// TIA Portal V16 export
// export: Created 2022-11-24T15:20:55.7439913Z, ExportSetting WithDefaults, DisplayName Totally Integrated Automation Portal, DisplayVersion V16 Update 6, DisplayName TIA Portal Version Control Interface, DisplayVersion V16 Update 2, DisplayName TIA Portal Openness, DisplayVersion V16 Update 6, DisplayName SINAMICS Startdrive Advanced, DisplayVersion V16 Update 5, DisplayName SINAMICS Startdrive G130, G150, S120, S150, SINAMICS MV, S210, DisplayVersion V16 Update 5, DisplayName SINAMICS Startdrive G110M, G120, G120C, G120D, G120P, G115D, DisplayVersion V16 Update 5, DisplayName STEP 7 Professional, DisplayVersion V16 Update 6, DisplayName STEP 7 Safety, DisplayVersion V16, DisplayName WinCC Advanced, DisplayVersion V16 Update 6
FUNCTION "FC62_PreStretchPGSAoutPWM" : Void   // FC62, LAD
{ S7_Optimized_Access := 'FALSE' }
AUTHOR : PaZan
VERSION : 0.1
// stored: AutoNumber false, IsIECCheckEnabled false, SetENOAutomatically false, UDAEnableTagReadback false
BEGIN

REGION Network 1: copy parameter for scale value % prestretch
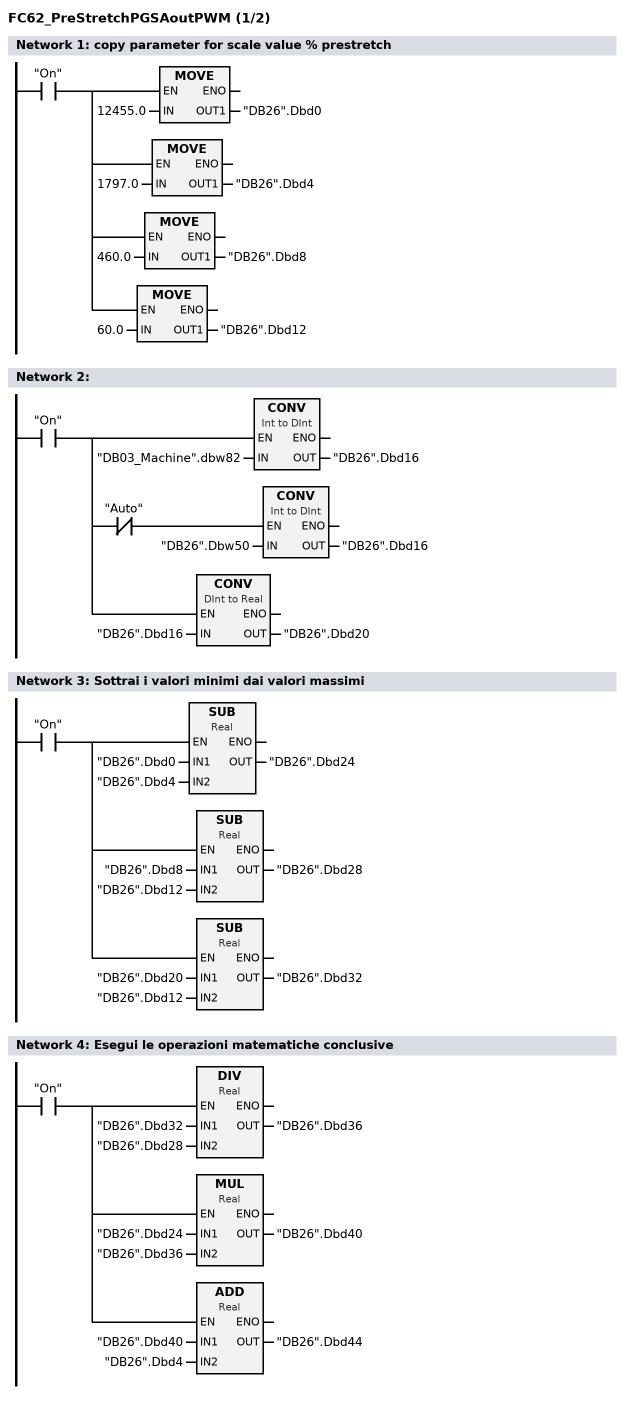
   RUNG wire#powerrail
      Contact( "On" )
      wire#w1
      { S7_GenerateENO := "TRUE" } Move(in := 12455.0, out1 => "DB26".Dbd0)
   END_RUNG
   RUNG wire#w1
      { S7_GenerateENO := "TRUE" } Move(in := 1797.0, out1 => "DB26".Dbd4)
   END_RUNG
   RUNG wire#w1
      { S7_GenerateENO := "TRUE" } Move(in := 460.0, out1 => "DB26".Dbd8)
   END_RUNG
   RUNG wire#w1
      { S7_GenerateENO := "TRUE" } Move(in := 60.0, out1 => "DB26".Dbd12)
   END_RUNG
   // the same network as SCL:
   IF "On" THEN
       "DB26".Dbd0 := 12455.0;
       "DB26".Dbd4 := 1797.0;
       "DB26".Dbd8 := 460.0;
       "DB26".Dbd12 := 60.0;
   END_IF;
END_REGION

REGION Network 2
   RUNG wire#powerrail
      Contact( "On" )
      wire#w1
      { S7_Templates := "[SrcType := Int, DestType := DInt]"; S7_GenerateENO := "TRUE" } Convert(in := "DB03_Machine".dbw82, out => "DB26".Dbd16)
   END_RUNG
   RUNG wire#w1
      I_Contact( "Auto" )
      { S7_Templates := "[SrcType := Int, DestType := DInt]"; S7_GenerateENO := "TRUE" } Convert(in := "DB26".Dbw50, out => "DB26".Dbd16)
   END_RUNG
   RUNG wire#w1
      { S7_Templates := "[SrcType := DInt, DestType := Real]"; S7_GenerateENO := "TRUE" } Convert(in := "DB26".Dbd16, out => "DB26".Dbd20)
   END_RUNG
   // the same network as SCL:
   IF "On" THEN "DB26".Dbd16 := INT_TO_DINT("DB03_Machine".dbw82); END_IF;
   IF "On" AND NOT "Auto" THEN "DB26".Dbd16 := INT_TO_DINT("DB26".Dbw50); END_IF;
   IF "On" THEN "DB26".Dbd20 := DINT_TO_REAL("DB26".Dbd16); END_IF;
END_REGION

REGION Network 3: Sottrai i valori minimi dai valori massimi
   RUNG wire#powerrail
      Contact( "On" )
      wire#w1
      { S7_Templates := "SrcType := Real"; S7_GenerateENO := "TRUE" } Sub(in1 := "DB26".Dbd0, in2 := "DB26".Dbd4, out => "DB26".Dbd24)
   END_RUNG
   RUNG wire#w1
      { S7_Templates := "SrcType := Real"; S7_GenerateENO := "TRUE" } Sub(in1 := "DB26".Dbd8, in2 := "DB26".Dbd12, out => "DB26".Dbd28)
   END_RUNG
   RUNG wire#w1
      { S7_Templates := "SrcType := Real"; S7_GenerateENO := "TRUE" } Sub(in1 := "DB26".Dbd20, in2 := "DB26".Dbd12, out => "DB26".Dbd32)
   END_RUNG
   // the same network as SCL:
   IF "On" THEN
       "DB26".Dbd24 := "DB26".Dbd0 - "DB26".Dbd4;
       "DB26".Dbd28 := "DB26".Dbd8 - "DB26".Dbd12;
       "DB26".Dbd32 := "DB26".Dbd20 - "DB26".Dbd12;
   END_IF;
END_REGION

REGION Network 4: Esegui le operazioni matematiche conclusive
   RUNG wire#powerrail
      Contact( "On" )
      wire#w1
      { S7_Templates := "SrcType := Real"; S7_GenerateENO := "TRUE" } Div(in1 := "DB26".Dbd32, in2 := "DB26".Dbd28, out => "DB26".Dbd36)
   END_RUNG
   RUNG wire#w1
      { S7_Templates := "SrcType := Real"; S7_GenerateENO := "TRUE" } Mul(in1 := "DB26".Dbd24, in2 := "DB26".Dbd36, out => "DB26".Dbd40)
   END_RUNG
   RUNG wire#w1
      { S7_Templates := "SrcType := Real"; S7_GenerateENO := "TRUE" } Add(in1 := "DB26".Dbd40, in2 := "DB26".Dbd4, out => "DB26".Dbd44)
   END_RUNG
   // the same network as SCL:
   IF "On" THEN
       "DB26".Dbd36 := "DB26".Dbd32 / "DB26".Dbd28;
       "DB26".Dbd40 := "DB26".Dbd24 * "DB26".Dbd36;
       "DB26".Dbd44 := "DB26".Dbd40 + "DB26".Dbd4;
   END_IF;
END_REGION

REGION Network 5: Trunc and copy value for pre-stretch in analogic out
   // PAW128
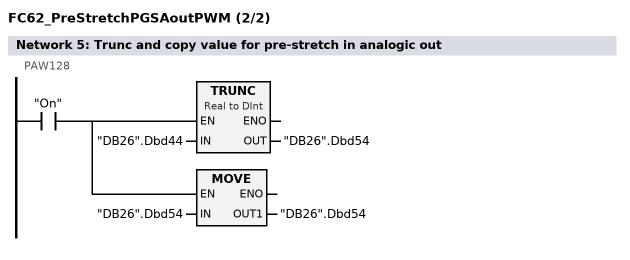
   RUNG wire#powerrail
      Contact( "On" )
      wire#w1
      { S7_Templates := "[SrcType := Real, DestType := DInt]"; S7_GenerateENO := "TRUE" } Trunc(in := "DB26".Dbd44, out => "DB26".Dbd54)
   END_RUNG
   RUNG wire#w1
      { S7_GenerateENO := "TRUE" } Move(in := "DB26".Dbd54, out1 => "DB26".Dbd54)
   END_RUNG
   // the same network as SCL:
   IF "On" THEN
       "DB26".Dbd54 := TRUNC("DB26".Dbd44);
       "DB26".Dbd54 := "DB26".Dbd54;
   END_IF;
END_REGION
END_FUNCTION
